Staubli VAL3: dataReset.pgx

program dataReset()
  local num ni
begin
  clearBuffer(sSocket1)
end
